# EPICS substitutions: vscode/appTest/test01App/Db/test03.substitutions
file test01.db {
    { IOCNAME=CCL_PS:IOC1, ABC=aaa }
    { IOCNAME=CCL_PS:IOC1, ABC=bbb }
}

file test01.db {
    pattern { IOCNAME,     ABC }
            { "",          "" }
            { CCL_PS:IOC1, bbb }
}
